// TIA Portal V20 export
FUNCTION_BLOCK "FB_AnalogOutput"   // FB33, SCL
{ S7_Optimized_Access := 'TRUE' }
// stored: AutoNumber false, MemoryReserve 100, SetENOAutomatically false
   VAR_INPUT
      iLimitUp { ExternalAccessible := 'False'; ExternalVisible := 'False'; ExternalWritable := 'False'} : Real;   // Limit up real value
      iLimitDown { ExternalAccessible := 'False'; ExternalVisible := 'False'; ExternalWritable := 'False'} : Real;   // Limit down real value
      iMaxAIWordValue { ExternalAccessible := 'False'; ExternalVisible := 'False'; ExternalWritable := 'False'} : Real;   // Word analog output range
   END_VAR
   VAR_OUTPUT
      oValueHW { ExternalAccessible := 'False'; ExternalVisible := 'False'; ExternalWritable := 'False'} : Word;   // Value in word for PLC analog output
   END_VAR
   VAR
      sSWRealValue { ExternalAccessible := 'False'; ExternalVisible := 'False'; ExternalWritable := 'False'} : Real;
      sHWWordValue { ExternalAccessible := 'False'; ExternalVisible := 'False'; ExternalWritable := 'False'} : Word;
   END_VAR
   VAR_TEMP
      tValueSWInt : Int;   // Int value (conversion)
      tValueSWWord : Word;   // Word value to set as PLC analog output
      tRange : Real;   // Real value range
      tValueSWReal : Real;   // Real value in absolute
   END_VAR
BEGIN
   REGION Description header 
       //==================================================================================
       // POSALUX Swiss SA / (C) Copyright 2024
       //----------------------------------------------------------------------------------
       // Title: Analog output function
       // Comment/Function: This function handles analog value conversion AND scaling.  
       //                   It converts a real value to an integer value, then to a word
       //                   for the PLC's analog output. The function also performs scaling
       //                   based on specified limits.
       // Author: Gowsigan SRITHARAN
       // Engineering: TIA Portal v17
       //----------------------------------------------------------------------------------
       // Change log table:
       // Version  | Date     | Expert in charge | Changes applied
       // ---------|----------|------------------|-----------------------------------------
       // 00.00.01 | 20250106 | GSR              | First released version
       // =================================================================================
   END_REGION

   REGION Initialization
       #tValueSWReal := #sSWRealValue;
   END_REGION

   REGION Absolute Value Calculation and Scaling
       // Calculate range
       #tRange := #iLimitUp - #iLimitDown;

       // Scale the value
       #tValueSWReal := #tValueSWReal - #iLimitDown;
       #tValueSWReal := #tValueSWReal / #tRange;
       #tValueSWReal := #tValueSWReal * #iMaxAIWordValue;
   END_REGION

   REGION Real-to-Word Value Conversion
       // Convert REAL to INT
       #tValueSWInt := REAL_TO_INT(#tValueSWReal);

       // Convert INT to WORD
       #tValueSWWord := INT_TO_WORD(#tValueSWInt);

       // Assign output values
       #sHWWordValue := #tValueSWWord;
       #oValueHW := #tValueSWWord;
   END_REGION
END_FUNCTION_BLOCK
